PROGRAM MAIN
VAR
	Xts				  : XtsSystem('XTS ProcessingUnit 1');
	Movers			  : ARRAY[1..2] OF XtsMover[('Mover 1', 0, Xts), ('Mover 2', 0, Xts)];
	VirtualCollection : XtsMoverCollection;
	ReleaseTrigger	  : XtsPositionTrigger('Release Trigger', 0, VirtualCollection, Xts);
	VirtualMover	  : XtsMover('Virtual Mover', 0, Xts);
	WholeTrack		  : XtsZone('Whole Track', Xts.Movers, 0, 1500, Xts);
	MoveVelocity	  : XtsMoverMoveVelocity;
	Halt			  : XtsMoverHalt;
	tmp AT %I*		  : UINT;
	State			  : UDINT;
	Hmi				  : XtsBasicHmi<3, 1, 3, 1>('Hmi', Xts);

	//
	startVirtualPosition : LREAL;
	SetPosition			 : MC_SetPosition;
	MoveToPos			 : ARRAY[1..2] OF MC_MoveAbsolute;
	GearIn				 : ARRAY[1..2] OF MC_GearIn;
	PhaseAxis			 : ARRAY[1..2] OF MC_PhasingRelative;
	OpenCloseDistance	 : LREAL := 60;
	commandedPosition	 : ARRAY[1..2] OF LREAL;
	Gap					 : LREAL := 115;
	newPosition			 : LREAL;

	//
	PickupPosition : LREAL := 875;
	DelayTimer	   : TON;
	PrePickupTime  : TIME  := T#5S;
	PostPickupTIme : TIME  := T#2S;
	ProductSpeed   : LREAL := 400;
	OpenVelocity   : LREAL := 600;

	//Reversing Sequence
	stopReversing : BOOL;
	DwellTime	  : TIME := T#3S;
	DwellTimer	  : TON;
	Pos1		  : LREAL := 750;
	Pos2		  : LREAL := 1000;
	godotHmi	  : GodotHmi(Movers[1]);

	//BallScrew Sample
	SyncTrigger	  : XtsPositionTrigger('SyncTrigger', 750, VirtualCollection, Xts);
	DesyncTrigger : XtsPositionTrigger('DesyncTrigger', 1000, VirtualCollection, Xts);
	FeedAxis	  : AXIS_REF;
	Feeder		  : AxisPTP('Feeder', FeedAxis);
	DeSyncedSpeed : LREAL := 200;
	AxisSpeed	  : LREAL := 200;
	Mover		  : I_XtsMover;
	Pitch		  : LREAL := 50;
	SyncPosition  : LREAL := 1100;
	_NextPocket	  : UDINT;

	// Cam Generator
	CurveComp	   : CamBuild;
	MoverCurveComp : CamCurveComp;
	MultiCamComp   : SplitCamBuild;
	MultiCamTest   : SplitCamRun;
END_VAR

IF NOT Xts.Initialized OR NOT Feeder.Initialized THEN
	Feeder.Initialize();
	Xts.Initialize();
	Xts.Parameters.Velocity		 := 200;
	Xts.Parameters.Acceleration	 := 5_000;
	Xts.Parameters.Deceleration	 := 5_000;
	Xts.Parameters.Jerk			 := 100_000;
	Xts.Parameters.Gap			 := 100;
	VirtualMover.VirtualMover	 := TRUE;
	Movers[1].ManualGroupControl := TRUE;
	Movers[2].ManualGroupControl := TRUE;
	Hmi.BuildHMI();
	IF VirtualCollection.IsEmpty THEN
		VirtualCollection.AddItem(VirtualMover);
	END_IF

	RETURN;
END_IF

CASE State OF
	0:
	1:
		Xts.Reset();
		Xts.ResetMovers();
		State := 0;

	5:
		Xts.Utility.SetConfiguredDetectionCount(Xts.Utility.GetDetectedMoverCount());
		State := 1;

	10:
		Xts.Enable();
		IF Xts.Enabled THEN
			State := 50;
		END_IF

	20:
		Xts.Disable();
		IF NOT Xts.Enabled THEN
			State := 0;
		END_IF

	60:
		MoveVelocity.CopyParametersFrom(Xts.Parameters);
		MoveVelocity.ExecuteOn(Xts);
		State := 50;

	61:
		Halt.CopyParametersFrom(Xts.Parameters);
		Halt.ExecuteOn(Xts);
		State := 50;

	70:
		MoveVelocity.CopyParametersFrom(Xts.Parameters);
		MoveVelocity.ExecuteOn(VirtualMover);
		State := 50;

	71:
		Halt.CopyParametersFrom(Xts.Parameters);
		Halt.ExecuteOn(VirtualMover);
		State := 50;

	100:
		IF Xts.Utility.GetMoverIdDetectionState() <> MoverIdDetectionStateEnum.Valid THEN
			State := 101;
		ELSE
			State := 111;
		END_IF

	101:
		Xts.Enable();
		IF Xts.Enabled THEN
			State := 102;
		END_IF

	102:
		Xts.Disable();
		IF NOT Xts.Enabled THEN
			State := 100;
		END_IF

	110:
		Xts.Disable();
		IF NOT Xts.Enabled THEN
			State := 111;
		END_IF

	111:
		//startVirtualPosition := (Movers[2].Position - Movers[1].Position) / 2 + Movers[1].Position;
		startVirtualPosition := 59;
		SetPosition(Axis := VirtualMover.Axis, Position := startVirtualPosition, Execute := TRUE);
		IF SetPosition.Done OR SetPosition.Error THEN
			State := 120;
			SetPosition(Axis := VirtualMover.Axis, Execute := FALSE);
		END_IF

	120:
		Xts.Enable();
		IF Xts.Enabled THEN
			State := 122;
		END_IF

	121:
		VirtualMover.Parameters.CopyFrom(Xts.Parameters);
		VirtualMover.Parameters.Gap := 0;
		VirtualMover.MoveToPosition(VirtualMover.Position);
		Movers[1].Parameters.CopyFrom(Xts.Parameters);
		Movers[2].Parameters.CopyFrom(Xts.Parameters);
		commandedPosition[1] := startVirtualPosition - Gap;
		commandedPosition[2] := startVirtualPosition + Gap;
		MoveToPos[1](Axis		  := Movers[1].Axis,
					 Execute	  := TRUE,
					 Position	  := commandedPosition[1],
					 Velocity	  := 300,
					 Acceleration := 5000,
					 Deceleration := 5000,
					 Jerk		  := 100000);

		MoveToPos[2](Axis		  := Movers[2].Axis,
					 Execute	  := TRUE,
					 Position	  := commandedPosition[2],
					 Velocity	  := 300,
					 Acceleration := 5000,
					 Deceleration := 5000,
					 Jerk		  := 100000);

		IF MoveToPos[1].Error OR MoveToPos[2].Error OR (MoveToPos[1].Done AND MoveToPos[2].Done) THEN
			MoveToPos[1](Axis := Movers[1].Axis, Execute := FALSE);
			MoveToPos[2](Axis := Movers[2].Axis, Execute := FALSE);
			State := 125;
		END_IF

	122:
		VirtualMover.Parameters.CopyFrom(Xts.Parameters);
		VirtualMover.Parameters.Gap := 0;
		VirtualMover.MoveToPosition(VirtualMover.Position);
		Movers[1].Parameters.CopyFrom(Xts.Parameters);
		Movers[2].Parameters.CopyFrom(Xts.Parameters);
		commandedPosition[1] := 115;
		commandedPosition[2] := commandedPosition[1] - Gap;
		MoveToPos[1](Axis		  := Movers[1].Axis,
					 Execute	  := TRUE,
					 Position	  := commandedPosition[1] + TRUNC(Movers[1].Axis.NcToPlc.ActPos / 1500.0) * 1500,
					 Velocity	  := 300,
					 Acceleration := 5000,
					 Deceleration := 5000,
					 Jerk		  := 100000);

		MoveToPos[2](Axis		  := Movers[2].Axis,
					 Execute	  := TRUE,
					 Position	  := commandedPosition[2] + TRUNC(Movers[1].Axis.NcToPlc.ActPos / 1500.0) * 1500,
					 Velocity	  := 300,
					 Acceleration := 5000,
					 Deceleration := 5000,
					 Jerk		  := 100000);

		IF MoveToPos[1].Error OR MoveToPos[2].Error OR (MoveToPos[1].Done AND MoveToPos[2].Done) THEN
			MoveToPos[1](Axis := Movers[1].Axis, Execute := FALSE);
			MoveToPos[2](Axis := Movers[2].Axis, Execute := FALSE);
			State := 125;
		END_IF

	125:
		GearIn[1](Master	   := VirtualMover.Axis,
				  Slave		   := Movers[1].Axis,
				  Execute	   := TRUE,
				  Acceleration := 10_000,
				  Deceleration := 10_000,
				  Jerk		   := 100_000);

		GearIn[2](Master	   := VirtualMover.Axis,
				  Slave		   := Movers[2].Axis,
				  Execute	   := FALSE,
				  Acceleration := 10_000,
				  Deceleration := 10_000,
				  Jerk		   := 100_000);

		IF GearIn[1].InGear (*AND GearIn[2].InGear *) THEN
			GearIn[1](Master := VirtualMover.Axis, Slave := Movers[1].Axis, Execute := FALSE);
			GearIn[2](Master := VirtualMover.Axis, Slave := Movers[2].Axis, Execute := FALSE);
			State := 150;
		END_IF

	130:
		VirtualMover.Parameters.CopyFrom(Xts.Parameters);
		VirtualMover.MoveToPosition(newPosition, XtsCore.Tc3_Mc3Definitions.MC_DIRECTION.mcDirectionShortestWay);
		State := 150;

	135:
		VirtualMover.Parameters.CopyFrom(Xts.Parameters);
		VirtualMover.MoveVelocity(Xts.Parameters.Velocity);
		State := 150;

	136:
		VirtualMover.Halt(Xts.Parameters.Deceleration, Xts.Parameters.Gap);
		State := 150;

	//Reversing Sequence 150-155
	160:
		VirtualMover.Parameters.CopyFrom(Xts.Parameters);
		VirtualMover.MoveToPosition(Pos1, XtsCore.Tc3_Mc3Definitions.MC_DIRECTION.mcDirectionShortestWay);
		State := 161;

	161:
		DwellTimer(IN := VirtualMover.InPosition, PT := DwellTime);
		IF DwellTimer.Q THEN
			DwellTimer(IN := FALSE);
			State := 162;
		END_IF

	162:
		VirtualMover.Parameters.CopyFrom(Xts.Parameters);
		VirtualMover.MoveToPosition(Pos2, XtsCore.Tc3_Mc3Definitions.MC_DIRECTION.mcDirectionShortestWay);
		State := 163;

	163:
		DwellTimer(IN := VirtualMover.InPosition, PT := DwellTime);
		IF DwellTimer.Q THEN
			DwellTimer(IN := FALSE);
			State := 164;
		END_IF

	164:
		IF stopReversing THEN
			stopReversing := FALSE;
			State		  := 150;
		ELSE
			State := 160;
		END_IF

	140:
		PhaseAxis[1](Master		  := VirtualMover.Axis,
					 Slave		  := Movers[1].Axis,
					 Execute	  := TRUE,
					 PhaseShift	  := OpenCloseDistance,
					 Velocity	  := Xts.Parameters.Velocity * 1.2,
					 Acceleration := 10_000,
					 Deceleration := 10_000,
					 Jerk		  := 100_000);

		PhaseAxis[2](Master		  := VirtualMover.Axis,
					 Slave		  := Movers[2].Axis,
					 Execute	  := FALSE,
					 PhaseShift	  := OpenCloseDistance,
					 Velocity	  := Xts.Parameters.Velocity * 1.2,
					 Acceleration := 10_000,
					 Deceleration := 10_000,
					 Jerk		  := 100_000);

		IF PhaseAxis[1].Error OR PhaseAxis[1].Done THEN
			PhaseAxis[1](Master := VirtualMover.Axis, Slave := Movers[1].Axis, Execute := FALSE);
			PhaseAxis[2](Master := VirtualMover.Axis, Slave := Movers[2].Axis, Execute := FALSE);
			State := 150;
		END_IF

	200:
		//Move to pick up position

		//Wait at pickup up position for PickupTime

		//Phase to close and pickup the ball

		//Move velocity

		//Trigger Active, tell Mover[1] to phase open distance
		//Phase Done, go back to repeat
		VirtualMover.MoveToPosition(PickupPosition);
		IF NOT VirtualMover.CurrentTask.Busy AND VirtualMover.InPosition THEN
			State := 210;
		END_IF

	210:
		DelayTimer(IN := TRUE, PT := PrePickupTime);
		IF DelayTimer.Q THEN
			DelayTimer(IN := FALSE);
			State := 211;
		END_IF

	211:
		PhaseAxis[1](Master		  := VirtualMover.Axis,
					 Slave		  := Movers[1].Axis,
					 Execute	  := TRUE,
					 PhaseShift	  := OpenCloseDistance,
					 Velocity	  := Xts.Parameters.Velocity * 1.2,
					 Acceleration := 10_000,
					 Deceleration := 10_000,
					 Jerk		  := 100_000);

		IF PhaseAxis[1].Error OR PhaseAxis[1].Done THEN
			PhaseAxis[1](Master := VirtualMover.Axis, Slave := Movers[1].Axis, Execute := FALSE);
			State := 212;
		END_IF

	212:
		DelayTimer(IN := TRUE, PT := PostPickupTime);
		IF DelayTimer.Q THEN
			DelayTimer(IN := FALSE);
			VirtualMover.MoveVelocity(ProductSpeed);
			State := 213;
		END_IF

	213:
		IF ReleaseTrigger.MoverIsPresent THEN
			ReleaseTrigger.GetMover();
			State := 220;
		END_IF

	220:
		PhaseAxis[1](Master		  := VirtualMover.Axis,
					 Slave		  := Movers[1].Axis,
					 Execute	  := TRUE,
					 PhaseShift	  := -OpenCloseDistance,
					 Velocity	  := OpenVelocity,
					 Acceleration := 10_000,
					 Deceleration := 10_000,
					 Jerk		  := 100_000);

		IF PhaseAxis[1].Error OR PhaseAxis[1].Done THEN
			PhaseAxis[1](Master := VirtualMover.Axis, Slave := Movers[1].Axis, Execute := FALSE);
			State := 200;
		END_IF

	//Start of the BallScrew Sample Code
	300:
		//Set Master Position to 0
		Feeder.Home();
		IF NOT Feeder.Busy THEN
			State := 301;
		END_IF

	301:
		//Enable Master
		Feeder.Enable();
		IF Feeder.Enabled THEN
			State := 302;
		END_IF

	302:
		//enable the PosTrigger
		SyncTrigger.Enable();
		IF SyncTrigger.Enabled THEN
			State := 303;
			SyncTrigger.MoverQueue.Clear();
		END_IF

	303:
		//MoveVelocity on Master
		VirtualMover.MoveVelocity(DeSyncedSpeed);
		Feeder.MoveVelocity(AxisSpeed);
		State := 305;

	305:
		_NextPocket := DINT_TO_UDINT(TRUNC(Feeder.SetPosition / Pitch) + 1);
		//Monitor Trigger
		IF SyncTrigger.MoverIsPresent THEN
			Mover														  := SyncTrigger.GetMover();
			Mover.Parameters.Velocity									  := AxisSpeed * 2;
			Mover.Parameters.Acceleration								  := 10_000;
			Mover.Parameters.Deceleration								  := 10_000;
			Mover.Parameters.Jerk										  := 100_000;
			Mover.Parameters.SyncAxis.Options_CA.DirectionReversalAllowed := FALSE;
			Mover.Parameters.SyncAxis.SyncMode							  := XtsCore.Tc3_McCollisionAvoidance.MC_SYNC_MODE.mcSyncModePositive;
			Mover.SyncToAxis(Master := FeedAxis, MasterSyncPosition := _NextPocket * Pitch, SlaveSyncPosition := SyncPosition); //TOOD: Fix Position calcs
		END_IF

		IF DeSyncTrigger.MoverIsPresent THEN
			Mover := DeSyncTrigger.GetMover();
			Mover.MoveVelocity(DeSyncedSpeed);
		END_IF

	310:
		//Disable Trigger
		SyncTrigger.Disable();

		//Stop Master
		Feeder.Stop();
		IF Feeder.Stopped THEN
			State := 311;
		END_IF

	311:
		//Stop Zone
		VirtualMover.Halt(Xts.Parameters.Deceleration, Xts.Parameters.Gap);
		State := 312;

	312:
		IF NOT Halt.Busy THEN
			State := 313;
		END_IF

	313:
		Feeder.Disable();
		//Disable Master		
		IF NOT Feeder.Enabled THEN
			State := 150;
		END_IF

	401:
		CurveComp.Start();
		SetStep(State, 400);

	402:
		CurveComp.Reset();
		SetStep(State, 400);

	403:
		MultiCamComp.Start();
		SetStep(State, 400);

	404:
		MultiCamComp.Reset();
		SetStep(State, 400);

	410:
		MoverCurveComp.FrontMover	:= Movers[1];
		MoverCurveComp.RearMover	:= Movers[2];
		MoverCurveComp.VirtualMover := VirtualMover;
		MoverCurveComp.Start();
		NextMinorStep(State);

	411:
		IF NOT MoverCurveComp.Busy THEN
			SetStep(State, 400);
		END_IF

	412:
		MoverCurveComp.Reset();
		SetStep(State, 400);

	420:
		MultiCamTest.FrontMover	  := Movers[1];
		MultiCamTest.RearMover	  := Movers[2];
		MultiCamTest.VirtualMover := VirtualMover;
		MultiCamTest.Start();
		NextMinorStep(State);

	421:
		IF NOT MultiCamTest.Busy THEN
			SetStep(State, 400);
		END_IF

	422:
		MultiCamTest.Reset();
		SetStep(State, 400);
END_CASE

MultiCamComp.CyclicLogic();
MultiCamTest.CyclicLogic();
MoverCurveComp.CyclicLogic();
CurveComp.CyclicLogic();
Feeder.CyclicLogic();
godotHmi.CyclicLogic();
Xts.CyclicLogic();
Hmi.CyclicLogic();

END_PROGRAM

(* stored: Version 1.1.0.1, ProductVersion 3.1.4026.19
   POU MAIN: Id {ca052151-d944-4048-8176-ae57a0c29f6c}, SpecialFunc None *)
